// TIA Portal V17 export
// export: Created 2022-10-06T10:53:42.2067663Z, ExportSetting WithDefaults, DisplayName Totally Integrated Automation Portal, DisplayVersion V17, DisplayName TIA Portal Openness, DisplayVersion V17, DisplayName TIA Portal Version Control Interface, DisplayVersion V17, DisplayName SINAMICS Startdrive Advanced, DisplayVersion V17, DisplayName SINAMICS Startdrive G130, G150, S120, S150, SINAMICS MV, S210, DisplayVersion V17, DisplayName SINAMICS Startdrive G110M, G120, G120C, G120D, G120P, G115D, DisplayVersion V17, DisplayName STEP 7 Professional, DisplayVersion V17, DisplayName STEP 7 Safety, DisplayVersion V17, DisplayName WinCC Advanced, DisplayVersion V17
FUNCTION "Jaw" : Void   // FC1, LAD
{ S7_Optimized_Access := 'TRUE' }
VERSION : 0.1
// stored: AutoNumber true, IsIECCheckEnabled false, SetENOAutomatically false, UDAEnableTagReadback false
BEGIN

REGION Network 1
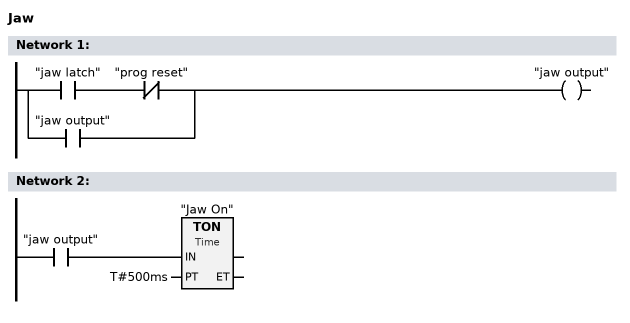
   RUNG wire#powerrail
      Contact( "jaw latch" )
      I_Contact( "prog reset" )
      wire#w1
      Coil( "jaw output" )
   END_RUNG
   RUNG wire#powerrail
      Contact( "jaw output" )
   END_RUNG wire#w1
   // the same network as SCL:
   "jaw output" := ("jaw latch" AND NOT "prog reset") OR "jaw output";
END_REGION

REGION Network 2
   RUNG wire#powerrail
      Contact( "jaw output" )
      { S7_Templates := "time_type := Time" } "Jaw On".TON(pt := T#500ms, et =>)
   END_RUNG
   // the same network as SCL:
   "Jaw On".TON(IN := "jaw output", PT := T#500ms);
END_REGION
END_FUNCTION
